PROGRAM B_1_1_PRG_Master_Station_1

VAR
	eState								: E_LeakTester_State;
	tonErrorReset						: TON;
	tonStationStopped					: TON;
	ctuErrorCounter						: CTU;
	rGoodStatistics						: R_TRIG;
	rBadStatistics						: R_TRIG;
	rEfficency							: STRING(510);
	
	bPersistentError					: BOOL;
	
	bEventsFlag							: ARRAY [0..100] OF BOOL;
/////////////////////////////////////////////////////////////////////////////////////I O/////////////////////////////////////////////////////////////////////////////////////	
	bStopped							: BOOL;
	bError								: BOOL;
	bReady								: BOOL;
	bDone								: BOOL;
	bPass								: BOOL;
	bFail								: BOOL;

	
END_VAR

VAR_INPUT	
	
	CMD									:ST_GeneralStationCMD;	
	
END_VAR

VAR_OUTPUT	
	
	STATUS								:ST_StationStatus;	
	
END_VAR

a_ACT_Ctrl_Station_1();
b_ACT_IO();
c_ACT_Statistics_Station_1();
d_ACT_Set_Events_Station_1();

ACTION a_ACT_Ctrl_Station_1:
/////////////////////////////////////////////////////////////////////////////////////UTILITIES/////////////////////////////////////////////////////////////////////////////////////
tonErrorReset( IN := (eState = E_LeakTester_State.RESET_ERROR), PT := T#500MS);
tonStationStopped( IN := bStopped, PT := T#1S);

ctuErrorCounter( CU := eState = E_LeakTester_State.RESET_ERROR, RESET := ((ctuErrorCounter.CV = 5) AND eState = E_LeakTester_State.PERSISTENT_ERROR), PV := 5, Q => bPersistentError);



/////////////////////////////////////////////////////////////////////////////////////CONDITIONS/////////////////////////////////////////////////////////////////////////////////////

IF (CMD.bAbort OR bError) AND ( eState			= E_LeakTester_State.HOMING OR
								eState			= E_LeakTester_State.READY OR
								eState			= E_LeakTester_State.MOVEMENT_A OR
								eState			= E_LeakTester_State.MOVEMENT_B OR
								eState			= E_LeakTester_State.MOVEMENT_C OR
								eState			= E_LeakTester_State.READY OR
								eState			= E_LeakTester_State.DONE) THEN
								
	eState						:= E_LeakTester_State.STOPPING;
	
END_IF



CASE eState OF
	
	E_LeakTester_State.ABORTED:
								IF CMD.bEnable AND NOT bError THEN
									eState						:= E_LeakTester_State.HOMING;
								ELSIF bError THEN
									eState						:= E_LeakTester_State.ERROR;
								END_IF
	
	E_LeakTester_State.HOMING:
								IF bReady THEN
									eState						:= E_LeakTester_State.RESET;
								END_IF
																
	E_LeakTester_State.RESET:
								stCycleDataStation1.bPass	:= FALSE;
								stCycleDataStation1.bFail	:= FALSE;
								
								eState						:= E_LeakTester_State.READY;
	E_LeakTester_State.READY:
								IF CMD.bExecute AND stStation1.Mov1 THEN
									eState						:= E_LeakTester_State.MOVEMENT_A;
								ELSIF CMD.bExecute AND stStation1.Mov2 THEN
									eState						:= E_LeakTester_State.MOVEMENT_B;
								ELSIF CMD.bExecute AND stStation1.Mov3 THEN
									eState						:= E_LeakTester_State.MOVEMENT_C;
								END_IF
	
	E_LeakTester_State.MOVEMENT_A:
								IF bDone AND stStation1.Mov1 THEN
									eState						:= E_LeakTester_State.DONE;
								END_IF
	
	E_LeakTester_State.MOVEMENT_B:
								IF bDone AND stStation1.Mov2 THEN
									eState						:= E_LeakTester_State.DONE;
								END_IF
	E_LeakTester_State.MOVEMENT_C:
								IF bDone AND stStation1.Mov3 THEN
									eState						:= E_LeakTester_State.DONE;
								END_IF
	E_LeakTester_State.DONE:
								IF  CMD.bReady THEN
									eState						:= E_LeakTester_State.RESULTS;
								END_IF	
								
	E_LeakTester_State.RESULTS:
								
								IF bPass THEN
									stCycleDataStation1.bPass	:= TRUE;
								ELSIF bFail THEN
								 	stCycleDataStation1.bFail	:= TRUE;
								END_IF
								
								IF  CMD.bEndCycle THEN
									eState						:= E_LeakTester_State.RESET;
								END_IF
								
/////////////////////////////////////////////////////////////////////////////////////RESET CMD/////////////////////////////////////////////////////////////////////////////////////			
	
	E_LeakTester_State.STOPPING: 
								IF tonStationStopped.Q THEN
									IF bError THEN
										eState						:= E_LeakTester_State.ERROR;
									ELSE eState						:= E_LeakTester_State.ABORTED;
									END_IF

								END_IF
	
	E_LeakTester_State.ERROR:
								IF NOT bError THEN
									eState						:= E_LeakTester_State.ABORTED;
								ELSE eState						:= E_LeakTester_State.RESET_ERROR;
								END_IF
	
	E_LeakTester_State.RESET_ERROR:
								IF tonErrorReset.Q AND NOT bPersistentError THEN
									eState						:= E_LeakTester_State.ERROR;
								ELSIF bPersistentError THEN
									eState						:= E_LeakTester_State.PERSISTENT_ERROR;
								END_IF
	
	E_LeakTester_State.PERSISTENT_ERROR:
								IF CMD.bReset THEN
									eState						:= E_LeakTester_State.ERROR;
								END_IF
	


							
						
								
													
								

ELSE eState := E_LeakTester_State.ABORTED;
	
END_CASE
/////////////////////////////////////////////////////////////////////////////////////STATUS/////////////////////////////////////////////////////////////////////////////////////

Status.bBusy				:= 	eState			= E_LeakTester_State.HOMING OR
								eState			= E_LeakTester_State.MOVEMENT_A OR
								eState			= E_LeakTester_State.MOVEMENT_B OR
								eState			= E_LeakTester_State.MOVEMENT_C OR
								eState			= E_LeakTester_State.STOPPING;
								
Status.bDone				:=	eState			= E_LeakTester_State.DONE;
											
Status.bError				:= 	(eState			= E_LeakTester_State.ERROR) OR 
								(eState			= E_LeakTester_State.RESET_ERROR) OR
								(eState			= E_LeakTester_State.PERSISTENT_ERROR);
								
Status.bReady				:= 	eState			= E_LeakTester_State.READY;

Status.bStopped				:= 	eState			= E_LeakTester_State.ABORTED OR
								eState			= E_LeakTester_State.READY OR
								eState			= E_LeakTester_State.ERROR OR
								eState			= E_LeakTester_State.RESET_ERROR;
END_ACTION

ACTION b_ACT_IO:
//bStopped								:=;
//bError								:=;
//bReady								:=;
//bDone
END_ACTION

ACTION c_ACT_Statistics_Station_1:
stStatisticsHMI[1].sName			:= 'Station 1';


rGoodStatistics( CLK := (stCycleDataStation1.bPass AND (eState = E_LeakTester_State.RESULTS)) OR bStatisticsTest[0]);
rBadStatistics( CLK := (stCycleDataStation1.bFail AND (eState = E_LeakTester_State.RESULTS)) OR bStatisticsTest[1]);

IF 	rGoodStatistics.Q THEN
	
	stStatisticsHMI[1].nGood		:= stStatisticsHMI[1].nGood + 1;
	stStatisticsHMI[1].nTotalGood	:= stStatisticsHMI[1].nTotalGood + 1;
	
END_IF
								
IF 	rBadStatistics.Q THEN
	
	stStatisticsHMI[1].nBad			:= stStatisticsHMI[1].nBad + 1;
	stStatisticsHMI[1].nTotalBad	:= stStatisticsHMI[1].nTotalBad + 1;
	
END_IF

IF stStatisticsHMI[1].bResetGood THEN
	stStatisticsHMI[1].nGood		:= 0;
END_IF

IF stStatisticsHMI[1].bResetBad THEN
	stStatisticsHMI[1].nBad			:= 0;
END_IF



IF (( stStatisticsHMI[1].nGood + stStatisticsHMI[1].nBad) <> 0) THEN
	
	rEfficency							:= LREAL_TO_FMTSTR(in := (DINT_TO_REAL(stStatisticsHMI[1].nGood) /( DINT_TO_REAL(stStatisticsHMI[1].nGood) + DINT_TO_REAL(stStatisticsHMI[1].nBad))) * 100.0,iPrecision := 2, bRound := TRUE);
	stStatisticsHMI[1].nEfficency		:= CONCAT(STR1 := '%', STR2 := (rEfficency));

ELSE stStatisticsHMI[1].nEfficency		:= CONCAT(STR1 := '%', STR2 := (DINT_TO_STRING(0)));
	
END_IF
END_ACTION

ACTION d_ACT_Set_Events_Station_1:
//IMMEDIATE FAULTS

stStationEvents[1].aEvents[0].bImmediateFault				:= TRUE;
stStationEvents[1].aEvents[0].bEventFlag					:= bEventsFlag[0];
stStationEvents[1].aEvents[0].bEventText					:= 'ST1 EVENT 0';
stStationEvents[1].aEvents[0].sSolution						:= 'Solution 1';


//CYCLE STOP FAULT

stStationEvents[1].aEvents[1].bCycleStopFault				:= TRUE;
stStationEvents[1].aEvents[1].bEventFlag					:= bEventsFlag[1];
stStationEvents[1].aEvents[1].bEventText					:= 'ST1 EVENT 1';
stStationEvents[1].aEvents[1].sSolution						:= 'Solution 2';


//CYCLE STOP REQUEST

stStationEvents[1].aEvents[2].bCycleStopRequest			:= TRUE;
stStationEvents[1].aEvents[2].bEventFlag					:= bEventsFlag[2];
stStationEvents[1].aEvents[2].bEventText					:= 'ST1 EVENT 2';
stStationEvents[1].aEvents[2].sSolution						:= '';

//Message

stStationEvents[1].aEvents[3].bMessage						:= TRUE;
stStationEvents[1].aEvents[3].bEventFlag					:= bEventsFlag[3];
stStationEvents[1].aEvents[3].bEventText					:= 'Message 3';
stStationEvents[1].aEvents[3].sSolution						:= '';
END_ACTION

END_PROGRAM

(* stored: Version 1.1.0.1, ProductVersion 3.1.4024.13
   POU B_1_1_PRG_Master_Station_1: Id {74fda7da-e1c3-493f-8c86-5902a8ab2668}, SpecialFunc None
   Action a_ACT_Ctrl_Station_1: Id {ce5dd8ea-9899-4a9f-bde8-defccc1c38a2}
   Action b_ACT_IO: Id {0f51cbd8-7d44-46ba-8ff2-5b85b0a3ce4b}
   Action c_ACT_Statistics_Station_1: Id {33f3666a-9a01-47bc-b17c-8cc705cb878c}
   Action d_ACT_Set_Events_Station_1: Id {e78af74f-1632-4c5a-a6d8-e4aea7d2a011} *)
